(*
Nazwa:			FB_JiesangActuatorEncoder
Opis:			Obsługa podnosnika Jiesang
Wersja:			v0.1
Data:			2018-10-10
Autor:			TW
Urzadzenia:		waga HBM
Konfiguracja:	
Info: 
- podlaczenie po RS485
*)

///!!!!!WAŻNE!!!!!!!!!!
///ABY ENKODER PRACOWAŁ POPRAWNIE TASK PLC MUSI BYĆ USTAWIONY NA 3ms!!!!!!!!!
///Wynika to z faktu że korzystamy ze zwykłych wejść cyfrowych a nie szybkich liczników!!!


FUNCTION_BLOCK FB_JiesangActuatorEncoder
VAR_INPUT
	bUpDirectionOut:BOOL;  	//Zmienna sterownika bezpośrednio sterująca siłownikiem w górę (zlinkowana z wyjściem sterownika)
	bDownDirectionOut:BOOL;	//Zmienna sterownika bezpośrednio sterująca siłownikiem w dół (zlinkowana z wyjsciem sterownika)
	bEncoderPulse:BOOL;		//Sygnał impulsów enkodera siłownika
	bHomingCancel:BOOL;		//Anulowanie bazowania enkodera
	bPositionSet:BOOL;		//Zmienna ustawia aktualną wartości pozycji zawartą w zmiennej 'nPositionOffset'
	rPositionOffset:REAL;		//Wartość do nadpisania aktualnej pozycji po ustawieniu wejścia 'AcbtorPositionSet'
	rPulseRatio:REAL;			//Przelicznik impulsów na mm  (pokonana_odleglosc_w_mm/ilość_impulsów)
	
	bOptionCoutingFalling : BOOL;  //Obliczenie spadania silnika
 END_VAR
VAR_OUTPUT
	bHomingDone:BOOL;
	lrActuatorPosition:LREAL:=-200;
	lrPulseRised:LREAL;
	lrPulseFalled:LREAL;
END_VAR
VAR
	tonOffDelay	:	TON;
rtEncoderPulse:R_TRIG;  //wykrywanie zbocza narastającego impulsu encodera
ftEncoderPulse:F_TRIG;  //wykrywanie zbocza opadającego impulsu encodera
rtActuatorPositionSet:R_TRIG;
bLastDirectionUp:BOOL;
rtHomingCancel: R_TRIG;
	cnt : INT;
END_VAR



//Kasowanie pozycjonowania enkodera
rtHomingCancel(CLK:=bHomingCancel,Q=>);
IF rtHomingCancel.Q THEN
	bHomingDone:=FALSE;
	lrActuatorPosition:=-200;
END_IF

//Jeśli na wejsciu pojawi sie ustawianie aktualnej pozycji enkodera
rtActuatorPositionSet(CLK:=bPositionSet,Q=>);
IF rtActuatorPositionSet.Q THEN
	lrActuatorPosition:=rPositionOffset;
	bHomingDone:=TRUE;
	lrPulseRised:=0;
	lrPulseFalled:=0;
END_IF


//Zapisywanie ostatniego kierunku ruchu siłownika
IF bUpDirectionOut AND NOT bDownDirectionOut THEN
	bLastDirectionUp:=TRUE;
ELSIF bDownDirectionOut AND NOT bUpDirectionOut THEN
	bLastDirectionUp:=FALSE;	
END_IF

//Wykrywanie zbocza pulsu enkodera
rtEncoderPulse(CLK:=bEncoderPulse,Q=>);
ftEncoderPulse(CLK:=bEncoderPulse,Q=>);

tonOffDelay(IN:= NOT bUpDirectionOut AND NOT bDownDirectionOut, PT:=T#2S);

IF NOT bOptionCoutingFalling THEN
	IF rtEncoderPulse.Q OR ftEncoderPulse.Q THEN
		IF bLastDirectionUp THEN
			lrActuatorPosition:=lrActuatorPosition+rPulseRatio;
		ELSE
			lrActuatorPosition:=lrActuatorPosition-rPulseRatio;
		END_IF	
	END_IF
ELSE
	IF (bUpDirectionOut OR bDownDirectionOut) THEN
		IF rtEncoderPulse.Q OR ftEncoderPulse.Q THEN
			IF bLastDirectionUp THEN
				lrActuatorPosition:=lrActuatorPosition+rPulseRatio;
			ELSE
				lrActuatorPosition:=lrActuatorPosition-rPulseRatio;
			END_IF	
		END_IF
	ELSIF (NOT tonOffDelay.Q AND (rtEncoderPulse.Q OR ftEncoderPulse.Q)) THEN
		lrActuatorPosition:=lrActuatorPosition-rPulseRatio;
		cnt:=cnt +1;
	END_IF	
END_IF

END_FUNCTION_BLOCK

(* stored: Version 1.1.0.1, ProductVersion 3.1.4026.13, FileIdentifier a9fdb915f0c6921976f93730131f7b322d161357, FileSignature 759cd1fe615a5dfbb0aa26c778d065b1cc1b109f4a5f5403bebca579cb1c89198c592faf8ad8f0cdd8d1e82717529c02325193fd6aad3362a03885b3fd5326d9238e08fc5cf6d2a6767ef8d963dfd095056664995abaaa2391400692b3d5846a9bb0c0220e317b390595aadbeaf5836a8fbd8fa530f10288fa1492db250f46c7e97cd59f29dcbde45904bc46d8420ea0b05cc233ea48811be8705ad1a1a89ba8b8e43387c635973b2eb621d93ab4fa94440f6e7df57da745d19c33d19f96a3c566bd9323e8d644dccdafae61614619743e009467d88d348872592017e2264b1dc45a0785f3c4575ece0dae97062ccfed507f304fc54422de3fd661cd990aa35e
   POU FB_JiesangActuatorEncoder: Id {7461489e-46af-4457-90ac-c616742deeff}, SpecialFunc None *)
